// TIA Portal V20 export
DATA_BLOCK "DB_Test_Water_Foutain"   // DB4
{ S7_Optimized_Access := 'TRUE' }
// stored: MemoryReserve 100
   VAR
      Star_Functional_Test : Bool;
      Reset_Functional_Test : Bool;
      Electrical_Current_Test_Approved : Bool;
      Visual_Test_Approved_PLC : Bool;
   END_VAR
BEGIN
END_DATA_BLOCK
